TYPE T_TypeClass : __SYSTEM.TYPE_CLASS; END_TYPE

(* stored: Version 1.1.0.1
   DUT T_TypeClass: Id {7c2ddb7a-1f65-07a9-1274-2c2883426fbb} *)
